(* CODESYS project Gateway_MLP_Validation.ecp

Project tree, tasks and I/O mapping:
  Steuerung : 750-8202 PFC200 2ETH RS, WAGO, order no. 0750-8202, version 5.15.4.20
    application Application
      libraries: ; Energy Edge Library, 3.5.16.10 (Zittau_Goerlitz University of Applied Sciences - IPM)
      task MLPinference (cyclic, interval 5 ms, priority 4) calls MLPinference
      Symbols
      program MLPinference [ST]
      function block WineTestMLP_3Layer [ST]
      function block WineTestMLP_2Layer [ST]
      function block WineTestMLP_1Layer [ST]
    Kbus : Kbus, WAGO, version 1.4.0.2
        unmapped channels: K-BUS diagnostics
    MODBUS
      MODBUS : MODBUS, WAGO, order no. n/a, version 1.1.1.15
    Serial
      COM1 : COM1, WAGO, version 0.0.0.19
*)

// Steuerung/Application/MLPinference
PROGRAM MLPinference
VAR
	// Seperate Inputs, since writen on MLP inputs via OPC UA fails

	inMLP1: ARRAY[1..11] OF REAL;
	inMLP2: ARRAY[1..11] OF REAL;	
	inMLP3: ARRAY[1..11] OF REAL;		

	MLP1: WineTestMLP_1Layer;
	MLP2: WineTestMLP_2Layer;
	MLP3: WineTestMLP_3Layer;
	
	recalculate: BOOL:=False;

END_VAR

IF recalculate THEN
	MLP1(in_1:=inMLP1[1], in_2:=inMLP1[2], in_3:=inMLP1[3], in_4:=inMLP1[4],
         in_5:=inMLP1[5], in_6:=inMLP1[6], in_7:=inMLP1[7], in_8:=inMLP1[8],
         in_9:=inMLP1[9], in_10:=inMLP1[10], in_11:=inMLP1[11]);
	MLP2(in_1:=inMLP2[1], in_2:=inMLP2[2], in_3:=inMLP2[3], in_4:=inMLP2[4],
         in_5:=inMLP2[5], in_6:=inMLP2[6], in_7:=inMLP2[7], in_8:=inMLP2[8],
         in_9:=inMLP2[9], in_10:=inMLP2[10], in_11:=inMLP2[11]);
	MLP3(in_1:=inMLP3[1], in_2:=inMLP3[2], in_3:=inMLP3[3], in_4:=inMLP3[4],
         in_5:=inMLP3[5], in_6:=inMLP3[6], in_7:=inMLP3[7], in_8:=inMLP3[8],
         in_9:=inMLP3[9], in_10:=inMLP3[10], in_11:=inMLP3[11]);
	recalculate := FALSE;
END_IF;

END_PROGRAM

// Steuerung/Application/WineTestMLP_1Layer
FUNCTION_BLOCK WineTestMLP_1Layer

VAR_INPUT
    in_1: REAL;
    in_2: REAL;
    in_3: REAL;
    in_4: REAL;
    in_5: REAL;
    in_6: REAL;
    in_7: REAL;
    in_8: REAL;
    in_9: REAL;
    in_10: REAL;
    in_11: REAL;
END_VAR

VAR
(* input array *)
    input: ARRAY[1..11] OF REAL;

(* hidden layer *)
(* Layer 1 *)
(* Neurons *)
    neuron_1_1: EEL.Neuron := (weights:=ADR(weights_1_1), bias:=(dw:=16#3f53bbb2), output:=0.0);
    neuron_1_2: EEL.Neuron := (weights:=ADR(weights_1_2), bias:=(dw:=16#3e774c91), output:=0.0);
    neuron_1_3: EEL.Neuron := (weights:=ADR(weights_1_3), bias:=(dw:=16#3f1b8655), output:=0.0);
    neuron_1_4: EEL.Neuron := (weights:=ADR(weights_1_4), bias:=(dw:=16#3f3931a5), output:=0.0);
    neuron_1_5: EEL.Neuron := (weights:=ADR(weights_1_5), bias:=(dw:=16#bd22504d), output:=0.0);
    neuron_1_6: EEL.Neuron := (weights:=ADR(weights_1_6), bias:=(dw:=16#3fcfd5a5), output:=0.0);
    neuron_1_7: EEL.Neuron := (weights:=ADR(weights_1_7), bias:=(dw:=16#3f154126), output:=0.0);
    neuron_1_8: EEL.Neuron := (weights:=ADR(weights_1_8), bias:=(dw:=16#bd8d8525), output:=0.0);
    neuron_1_9: EEL.Neuron := (weights:=ADR(weights_1_9), bias:=(dw:=16#3eede2e5), output:=0.0);
    neuron_1_10: EEL.Neuron := (weights:=ADR(weights_1_10), bias:=(dw:=16#bea8523e), output:=0.0);
    neuron_1_11: EEL.Neuron := (weights:=ADR(weights_1_11), bias:=(dw:=16#3f69af07), output:=0.0);
    neuron_1_12: EEL.Neuron := (weights:=ADR(weights_1_12), bias:=(dw:=16#3f1f30b5), output:=0.0);
    neuron_1_13: EEL.Neuron := (weights:=ADR(weights_1_13), bias:=(dw:=16#bc74c74c), output:=0.0);
    neuron_1_14: EEL.Neuron := (weights:=ADR(weights_1_14), bias:=(dw:=16#be4313a3), output:=0.0);
    neuron_1_15: EEL.Neuron := (weights:=ADR(weights_1_15), bias:=(dw:=16#bd1f8833), output:=0.0);
    neuron_1_16: EEL.Neuron := (weights:=ADR(weights_1_16), bias:=(dw:=16#3fa90598), output:=0.0);
    neuron_1_17: EEL.Neuron := (weights:=ADR(weights_1_17), bias:=(dw:=16#3f770b9d), output:=0.0);
    neuron_1_18: EEL.Neuron := (weights:=ADR(weights_1_18), bias:=(dw:=16#be4901f0), output:=0.0);
    neuron_1_19: EEL.Neuron := (weights:=ADR(weights_1_19), bias:=(dw:=16#bec4c956), output:=0.0);
    neuron_1_20: EEL.Neuron := (weights:=ADR(weights_1_20), bias:=(dw:=16#3effbf04), output:=0.0);
    neuron_1_21: EEL.Neuron := (weights:=ADR(weights_1_21), bias:=(dw:=16#3edacf42), output:=0.0);
    neuron_1_22: EEL.Neuron := (weights:=ADR(weights_1_22), bias:=(dw:=16#3f23897f), output:=0.0);
    neuron_1_23: EEL.Neuron := (weights:=ADR(weights_1_23), bias:=(dw:=16#bea09cbd), output:=0.0);
    neuron_1_24: EEL.Neuron := (weights:=ADR(weights_1_24), bias:=(dw:=16#3dabf729), output:=0.0);
    neuron_1_25: EEL.Neuron := (weights:=ADR(weights_1_25), bias:=(dw:=16#3f37b6a8), output:=0.0);
    hl_1_neurons: ARRAY[1..25] OF EEL.Neuron := [neuron_1_1, neuron_1_2, neuron_1_3, neuron_1_4, neuron_1_5, neuron_1_6, neuron_1_7, neuron_1_8, neuron_1_9, neuron_1_10, neuron_1_11, neuron_1_12, neuron_1_13, neuron_1_14, neuron_1_15, neuron_1_16, neuron_1_17, neuron_1_18, neuron_1_19, neuron_1_20, neuron_1_21, neuron_1_22, neuron_1_23, neuron_1_24, neuron_1_25];
(* Layer *)
    hidden_layer_1: EEL.Layer := (neurons:=ADR(hl_1_neurons), nNeurons:=25,activation:=12, threshold:=0.0);


    hlArray: ARRAY[1..1] of EEL.Layer := [hidden_layer_1];

(* output layer *)
    neuron_out_1: EEL.Neuron := (weights:=ADR(weights_out_1), bias:=(dw:=16#3ed09339), output:=0.0);
    out_neurons: ARRAY[1..1] OF EEL.Neuron := [neuron_out_1];
    out_layer: EEL.Layer := (neurons:=ADR(out_neurons), nNeurons:=1,activation:=3, threshold:=0.0);

(* MLP representation *)
    MLP: EEL.ANN := (input:=ADR(input), hidden:=ADR(hlArray), output:=ADR(out_layer), nInput:=11, nHidden:=1);
END_VAR

VAR_OUTPUT
    out_1: REAL;
END_VAR

VAR CONSTANT
    weights_1_1: ARRAY[1..11] OF EEL.dwREAL := [(dw:=16#bd130818), (dw:=16#3e57655a), (dw:=16#be872a61), (dw:=16#bcbdb356), (dw:=16#bd1f8b54), (dw:=16#3d854569), (dw:=16#bd02e86e), (dw:=16#3e87b72d), (dw:=16#3e9c4398), (dw:=16#3d24639f), (dw:=16#be22c6a0)];
    weights_1_2: ARRAY[1..11] OF EEL.dwREAL := [(dw:=16#3e2ba454), (dw:=16#bdc5c676), (dw:=16#3e3ef366), (dw:=16#3dcf9a7e), (dw:=16#bc0609b7), (dw:=16#3e3a72e8), (dw:=16#3e11846d), (dw:=16#3dc9d7ec), (dw:=16#bdd3251f), (dw:=16#389c9ec9), (dw:=16#3e24acb1)];
    weights_1_3: ARRAY[1..11] OF EEL.dwREAL := [(dw:=16#be00d314), (dw:=16#be382183), (dw:=16#3d07dd70), (dw:=16#bceefbce), (dw:=16#3dd44598), (dw:=16#3e1c33b7), (dw:=16#39f62b92), (dw:=16#bd632ec5), (dw:=16#3e1fecc7), (dw:=16#3c2fda30), (dw:=16#3d905dc3)];
    weights_1_4: ARRAY[1..11] OF EEL.dwREAL := [(dw:=16#bddbb524), (dw:=16#be554af8), (dw:=16#bda919bf), (dw:=16#3d3703ce), (dw:=16#3d70f66f), (dw:=16#bd44988d), (dw:=16#be1d6751), (dw:=16#bde58050), (dw:=16#3e51e712), (dw:=16#3d526bf5), (dw:=16#3e8ed860)];
    weights_1_5: ARRAY[1..11] OF EEL.dwREAL := [(dw:=16#3cbcb2b7), (dw:=16#bd2ecc57), (dw:=16#3de0a9a4), (dw:=16#3d298d90), (dw:=16#3dca6477), (dw:=16#bd4ba2ee), (dw:=16#3db50ce4), (dw:=16#3de32933), (dw:=16#bdead230), (dw:=16#3e2f56eb), (dw:=16#bd958376)];
    weights_1_6: ARRAY[1..11] OF EEL.dwREAL := [(dw:=16#bd8e9c27), (dw:=16#bd91e1fa), (dw:=16#bd6ca227), (dw:=16#3d671770), (dw:=16#bddaab27), (dw:=16#3dcc26e8), (dw:=16#3db16b56), (dw:=16#3d64df82), (dw:=16#bd0246ff), (dw:=16#bbc6cdd1), (dw:=16#3c404dc6)];
    weights_1_7: ARRAY[1..11] OF EEL.dwREAL := [(dw:=16#3bdecc96), (dw:=16#3bcbe5da), (dw:=16#3d2b50a4), (dw:=16#ba119a45), (dw:=16#bc438bf5), (dw:=16#3cb34be6), (dw:=16#bbc305c3), (dw:=16#bd0c3413), (dw:=16#bc8fb328), (dw:=16#3d39dc50), (dw:=16#bc19c7e9)];
    weights_1_8: ARRAY[1..11] OF EEL.dwREAL := [(dw:=16#bd61108b), (dw:=16#3d89d629), (dw:=16#bda47e84), (dw:=16#3cf8d9d7), (dw:=16#3d37cc3c), (dw:=16#3d57bf62), (dw:=16#3d606ad1), (dw:=16#bca8c762), (dw:=16#bd42dc34), (dw:=16#3e484431), (dw:=16#bc7633b2)];
    weights_1_9: ARRAY[1..11] OF EEL.dwREAL := [(dw:=16#be2c82e7), (dw:=16#3a1d1415), (dw:=16#bc41a5cf), (dw:=16#be42033e), (dw:=16#3dfcefe9), (dw:=16#be5ec4aa), (dw:=16#3e7ccf63), (dw:=16#be80d6a0), (dw:=16#3dd53c26), (dw:=16#bd937622), (dw:=16#be0c4531)];
    weights_1_10: ARRAY[1..11] OF EEL.dwREAL := [(dw:=16#be06776f), (dw:=16#3dffc8fc), (dw:=16#be17173a), (dw:=16#3d96ac7d), (dw:=16#3dcdc910), (dw:=16#3e4becaa), (dw:=16#3e05caf9), (dw:=16#3d694d95), (dw:=16#3e4c0015), (dw:=16#3e0131af), (dw:=16#bb05edc3)];
    weights_1_11: ARRAY[1..11] OF EEL.dwREAL := [(dw:=16#baaef3be), (dw:=16#be9ec245), (dw:=16#be0b5339), (dw:=16#3e006836), (dw:=16#bde8412e), (dw:=16#bb3055bf), (dw:=16#be01a90f), (dw:=16#3e01d2dd), (dw:=16#bce8fa64), (dw:=16#3e055065), (dw:=16#3e91930c)];
    weights_1_12: ARRAY[1..11] OF EEL.dwREAL := [(dw:=16#3df17f00), (dw:=16#bdb42e39), (dw:=16#3d769b38), (dw:=16#bdc2bb37), (dw:=16#be4bf9f7), (dw:=16#3e8e241d), (dw:=16#bd767810), (dw:=16#be4b11ea), (dw:=16#3d8e9dea), (dw:=16#bc47063f), (dw:=16#3e94287b)];
    weights_1_13: ARRAY[1..11] OF EEL.dwREAL := [(dw:=16#bc31da42), (dw:=16#bbaf341a), (dw:=16#bd287b58), (dw:=16#3c0e403d), (dw:=16#3d6f0f74), (dw:=16#3ccf2a99), (dw:=16#3d13f55d), (dw:=16#3b114489), (dw:=16#bd69e583), (dw:=16#3dccc3e8), (dw:=16#bc997423)];
    weights_1_14: ARRAY[1..11] OF EEL.dwREAL := [(dw:=16#3daef258), (dw:=16#be002661), (dw:=16#bc943066), (dw:=16#3db41f9b), (dw:=16#bb69810f), (dw:=16#3ca87ded), (dw:=16#3e3b0260), (dw:=16#3be476e7), (dw:=16#bdc6e2b0), (dw:=16#be2a7ec6), (dw:=16#3e3a9ab0)];
    weights_1_15: ARRAY[1..11] OF EEL.dwREAL := [(dw:=16#bd4de256), (dw:=16#3db57c57), (dw:=16#bdd2bb51), (dw:=16#3b9a972b), (dw:=16#bce2314f), (dw:=16#bb6dffbb), (dw:=16#bcc0e659), (dw:=16#3d149e41), (dw:=16#bdd52a52), (dw:=16#3e109b63), (dw:=16#bc04c6f8)];
    weights_1_16: ARRAY[1..11] OF EEL.dwREAL := [(dw:=16#3d8a3290), (dw:=16#3e05ee2b), (dw:=16#3d3b6ae0), (dw:=16#be0a58bd), (dw:=16#3dcb868a), (dw:=16#3c0cf723), (dw:=16#bde642cb), (dw:=16#bde659ca), (dw:=16#be364439), (dw:=16#3c9d0bf7), (dw:=16#be07452f)];
    weights_1_17: ARRAY[1..11] OF EEL.dwREAL := [(dw:=16#3d877279), (dw:=16#3e6a124c), (dw:=16#3d89c304), (dw:=16#3e07ed15), (dw:=16#3e252507), (dw:=16#be3de3f9), (dw:=16#be1dd184), (dw:=16#be851a24), (dw:=16#be94df33), (dw:=16#3e2c25ab), (dw:=16#3e250f69)];
    weights_1_18: ARRAY[1..11] OF EEL.dwREAL := [(dw:=16#bdeffadc), (dw:=16#bbd445cd), (dw:=16#bd498081), (dw:=16#3d837042), (dw:=16#bc6897bc), (dw:=16#be0bb273), (dw:=16#bdd77bed), (dw:=16#3c2604ab), (dw:=16#3e0991f3), (dw:=16#be4156f8), (dw:=16#3d8961a7)];
    weights_1_19: ARRAY[1..11] OF EEL.dwREAL := [(dw:=16#be60b820), (dw:=16#3e21be27), (dw:=16#bde0895a), (dw:=16#3c9ac8a0), (dw:=16#bdb6ab4f), (dw:=16#be2dbcf9), (dw:=16#be5d9323), (dw:=16#bd8e68dc), (dw:=16#3e2a844a), (dw:=16#beabbf6f), (dw:=16#3d7e7c9e)];
    weights_1_20: ARRAY[1..11] OF EEL.dwREAL := [(dw:=16#bdcd5501), (dw:=16#be35d7ff), (dw:=16#3e303c6a), (dw:=16#be29afe9), (dw:=16#be26862a), (dw:=16#be71656f), (dw:=16#bd35a65b), (dw:=16#3e7fae89), (dw:=16#be4008df), (dw:=16#3c073f38), (dw:=16#be4e845b)];
    weights_1_21: ARRAY[1..11] OF EEL.dwREAL := [(dw:=16#3d390b1c), (dw:=16#bd115fab), (dw:=16#3d306b93), (dw:=16#3c9372fd), (dw:=16#3b0bcc82), (dw:=16#3d0683fc), (dw:=16#bbe2c3af), (dw:=16#3c862552), (dw:=16#bd4d01b2), (dw:=16#3c988d92), (dw:=16#bd2800f4)];
    weights_1_22: ARRAY[1..11] OF EEL.dwREAL := [(dw:=16#bbcb6e7b), (dw:=16#3e93875e), (dw:=16#be8d8ad9), (dw:=16#3e3f7533), (dw:=16#bc0ee5ac), (dw:=16#be08c27e), (dw:=16#3eac5c4a), (dw:=16#bd94b032), (dw:=16#3e0d7cf5), (dw:=16#be485a5c), (dw:=16#bd07ce5c)];
    weights_1_23: ARRAY[1..11] OF EEL.dwREAL := [(dw:=16#bd559301), (dw:=16#be76dd4c), (dw:=16#bda748ba), (dw:=16#3cbe5fca), (dw:=16#bdd581e7), (dw:=16#3e196f17), (dw:=16#3d4f4331), (dw:=16#be4c92fd), (dw:=16#bca87a69), (dw:=16#be99c89d), (dw:=16#3de3a266)];
    weights_1_24: ARRAY[1..11] OF EEL.dwREAL := [(dw:=16#3ce204a2), (dw:=16#3d2ce670), (dw:=16#bd0e1f3b), (dw:=16#bde02636), (dw:=16#bd87123b), (dw:=16#bd6a8d42), (dw:=16#bde5a62f), (dw:=16#3c966757), (dw:=16#3dbb1b95), (dw:=16#be1fc696), (dw:=16#3bb752e5)];
    weights_1_25: ARRAY[1..11] OF EEL.dwREAL := [(dw:=16#3e3c38e9), (dw:=16#bd7c99d2), (dw:=16#3d16c39b), (dw:=16#bc866f5f), (dw:=16#3da78cfd), (dw:=16#bc07e312), (dw:=16#bdfa3ecf), (dw:=16#3decc2d5), (dw:=16#bd90452f), (dw:=16#3d867e23), (dw:=16#3d921418)];
    weights_out_1: ARRAY[1..25] OF EEL.dwREAL :=[(dw:=16#3f0bce82), (dw:=16#3ebc1fc3), (dw:=16#3eb9c571), (dw:=16#3eb97b27), (dw:=16#be8543b2), (dw:=16#3f11acc1), (dw:=16#3e4f512a), (dw:=16#be29c067), (dw:=16#3ecb8c44), (dw:=16#beba6d21), (dw:=16#3f3f28dc), (dw:=16#3f133968), (dw:=16#bdc67fed), (dw:=16#be9ae745), (dw:=16#be2c1060), (dw:=16#3f06b65f), (dw:=16#3f0c39f2), (dw:=16#be8ef089), (dw:=16#bf00858d), (dw:=16#3f01f92b), (dw:=16#3e15fc18), (dw:=16#3edc4104), (dw:=16#beeb452e), (dw:=16#be4c2559), (dw:=16#3e87fc13)];
END_VAR

(* get inputs *)
input[1] := in_1;
input[2] := in_2;
input[3] := in_3;
input[4] := in_4;
input[5] := in_5;
input[6] := in_6;
input[7] := in_7;
input[8] := in_8;
input[9] := in_9;
input[10] := in_10;
input[11] := in_11;

(* MLP inference *)
EEL.CallANN(ANN:=MLP);

(* set outputs *)
out_1 := out_neurons[1].output;

END_FUNCTION_BLOCK

// Steuerung/Application/WineTestMLP_2Layer
FUNCTION_BLOCK WineTestMLP_2Layer

VAR_INPUT
    in_1: REAL;
    in_2: REAL;
    in_3: REAL;
    in_4: REAL;
    in_5: REAL;
    in_6: REAL;
    in_7: REAL;
    in_8: REAL;
    in_9: REAL;
    in_10: REAL;
    in_11: REAL;
END_VAR

VAR
(* input array *)
    input: ARRAY[1..11] OF REAL;

(* hidden layer *)
(* Layer 1 *)
(* Neurons *)
    neuron_1_1: EEL.Neuron := (weights:=ADR(weights_1_1), bias:=(dw:=16#3c825e3d), output:=0.0);
    neuron_1_2: EEL.Neuron := (weights:=ADR(weights_1_2), bias:=(dw:=16#bea43e80), output:=0.0);
    neuron_1_3: EEL.Neuron := (weights:=ADR(weights_1_3), bias:=(dw:=16#be707efb), output:=0.0);
    neuron_1_4: EEL.Neuron := (weights:=ADR(weights_1_4), bias:=(dw:=16#3e146b2a), output:=0.0);
    neuron_1_5: EEL.Neuron := (weights:=ADR(weights_1_5), bias:=(dw:=16#3f5269ab), output:=0.0);
    neuron_1_6: EEL.Neuron := (weights:=ADR(weights_1_6), bias:=(dw:=16#3f4f3302), output:=0.0);
    neuron_1_7: EEL.Neuron := (weights:=ADR(weights_1_7), bias:=(dw:=16#3f42e11b), output:=0.0);
    neuron_1_8: EEL.Neuron := (weights:=ADR(weights_1_8), bias:=(dw:=16#3f40ae65), output:=0.0);
    neuron_1_9: EEL.Neuron := (weights:=ADR(weights_1_9), bias:=(dw:=16#be83203b), output:=0.0);
    neuron_1_10: EEL.Neuron := (weights:=ADR(weights_1_10), bias:=(dw:=16#bea2b30d), output:=0.0);
    neuron_1_11: EEL.Neuron := (weights:=ADR(weights_1_11), bias:=(dw:=16#3f3500ff), output:=0.0);
    neuron_1_12: EEL.Neuron := (weights:=ADR(weights_1_12), bias:=(dw:=16#3eb84acd), output:=0.0);
    neuron_1_13: EEL.Neuron := (weights:=ADR(weights_1_13), bias:=(dw:=16#3f335357), output:=0.0);
    neuron_1_14: EEL.Neuron := (weights:=ADR(weights_1_14), bias:=(dw:=16#bdd40d48), output:=0.0);
    neuron_1_15: EEL.Neuron := (weights:=ADR(weights_1_15), bias:=(dw:=16#bd81df84), output:=0.0);
    neuron_1_16: EEL.Neuron := (weights:=ADR(weights_1_16), bias:=(dw:=16#bddf6ef8), output:=0.0);
    neuron_1_17: EEL.Neuron := (weights:=ADR(weights_1_17), bias:=(dw:=16#3e36da12), output:=0.0);
    neuron_1_18: EEL.Neuron := (weights:=ADR(weights_1_18), bias:=(dw:=16#3f045953), output:=0.0);
    neuron_1_19: EEL.Neuron := (weights:=ADR(weights_1_19), bias:=(dw:=16#3ed228f5), output:=0.0);
    neuron_1_20: EEL.Neuron := (weights:=ADR(weights_1_20), bias:=(dw:=16#3ed4b31e), output:=0.0);
    neuron_1_21: EEL.Neuron := (weights:=ADR(weights_1_21), bias:=(dw:=16#bde4ea74), output:=0.0);
    neuron_1_22: EEL.Neuron := (weights:=ADR(weights_1_22), bias:=(dw:=16#3ec57342), output:=0.0);
    neuron_1_23: EEL.Neuron := (weights:=ADR(weights_1_23), bias:=(dw:=16#3d34d29b), output:=0.0);
    neuron_1_24: EEL.Neuron := (weights:=ADR(weights_1_24), bias:=(dw:=16#3f80457c), output:=0.0);
    neuron_1_25: EEL.Neuron := (weights:=ADR(weights_1_25), bias:=(dw:=16#bdaa519e), output:=0.0);
    hl_1_neurons: ARRAY[1..25] OF EEL.Neuron := [neuron_1_1, neuron_1_2, neuron_1_3, neuron_1_4, neuron_1_5, neuron_1_6, neuron_1_7, neuron_1_8, neuron_1_9, neuron_1_10, neuron_1_11, neuron_1_12, neuron_1_13, neuron_1_14, neuron_1_15, neuron_1_16, neuron_1_17, neuron_1_18, neuron_1_19, neuron_1_20, neuron_1_21, neuron_1_22, neuron_1_23, neuron_1_24, neuron_1_25];
(* Layer *)
    hidden_layer_1: EEL.Layer := (neurons:=ADR(hl_1_neurons), nNeurons:=25,activation:=12, threshold:=0.0);

(* Layer 2 *)
(* Neurons *)
    neuron_2_1: EEL.Neuron := (weights:=ADR(weights_2_1), bias:=(dw:=16#bf209498), output:=0.0);
    neuron_2_2: EEL.Neuron := (weights:=ADR(weights_2_2), bias:=(dw:=16#beeab10d), output:=0.0);
    neuron_2_3: EEL.Neuron := (weights:=ADR(weights_2_3), bias:=(dw:=16#3f4d4c49), output:=0.0);
    neuron_2_4: EEL.Neuron := (weights:=ADR(weights_2_4), bias:=(dw:=16#3f306120), output:=0.0);
    neuron_2_5: EEL.Neuron := (weights:=ADR(weights_2_5), bias:=(dw:=16#3f02efd6), output:=0.0);
    hl_2_neurons: ARRAY[1..5] OF EEL.Neuron := [neuron_2_1, neuron_2_2, neuron_2_3, neuron_2_4, neuron_2_5];
(* Layer *)
    hidden_layer_2: EEL.Layer := (neurons:=ADR(hl_2_neurons), nNeurons:=5,activation:=12, threshold:=0.0);


    hlArray: ARRAY[1..2] of EEL.Layer := [hidden_layer_1, hidden_layer_2];

(* output layer *)
    neuron_out_1: EEL.Neuron := (weights:=ADR(weights_out_1), bias:=(dw:=16#3d255e43), output:=0.0);
    out_neurons: ARRAY[1..1] OF EEL.Neuron := [neuron_out_1];
    out_layer: EEL.Layer := (neurons:=ADR(out_neurons), nNeurons:=1,activation:=3, threshold:=0.0);

(* MLP representation *)
    MLP: EEL.ANN := (input:=ADR(input), hidden:=ADR(hlArray), output:=ADR(out_layer), nInput:=11, nHidden:=2);
END_VAR

VAR_OUTPUT
    out_1: REAL;
END_VAR

VAR CONSTANT
    weights_1_1: ARRAY[1..11] OF EEL.dwREAL := [(dw:=16#3c55f395), (dw:=16#3d97f889), (dw:=16#bdf2c0f1), (dw:=16#bd2fd6c7), (dw:=16#bb6cef76), (dw:=16#3cf182be), (dw:=16#bd105294), (dw:=16#3d93a886), (dw:=16#3dc68841), (dw:=16#3d14c557), (dw:=16#bde70111)];
    weights_1_2: ARRAY[1..11] OF EEL.dwREAL := [(dw:=16#3c87590b), (dw:=16#be179a25), (dw:=16#3dbbbc1f), (dw:=16#3df58434), (dw:=16#bb86d268), (dw:=16#3d6793f4), (dw:=16#3e2f66db), (dw:=16#bc1c4752), (dw:=16#bd771fa5), (dw:=16#3c9d340b), (dw:=16#3e2e124a)];
    weights_1_3: ARRAY[1..11] OF EEL.dwREAL := [(dw:=16#be1928ea), (dw:=16#bcb78dd7), (dw:=16#be1abcc7), (dw:=16#3cc4fb9c), (dw:=16#3e3e9e8c), (dw:=16#3dd5666e), (dw:=16#3e2c61fa), (dw:=16#bc51bda6), (dw:=16#bc0213e6), (dw:=16#3e843141), (dw:=16#bd86a7cd)];
    weights_1_4: ARRAY[1..11] OF EEL.dwREAL := [(dw:=16#bde9f6b3), (dw:=16#be864c9d), (dw:=16#bdd7d352), (dw:=16#3ddbbce3), (dw:=16#bd9425e1), (dw:=16#be54217c), (dw:=16#be8b1d76), (dw:=16#bead0200), (dw:=16#3e080905), (dw:=16#3e4c7713), (dw:=16#3edcc87a)];
    weights_1_5: ARRAY[1..11] OF EEL.dwREAL := [(dw:=16#be335363), (dw:=16#3e8dc1ea), (dw:=16#be03a942), (dw:=16#3bcf609d), (dw:=16#3e1897e6), (dw:=16#be4bf5fc), (dw:=16#bcd23276), (dw:=16#be42dff3), (dw:=16#3d43abaf), (dw:=16#393a1b60), (dw:=16#3d785a49)];
    weights_1_6: ARRAY[1..11] OF EEL.dwREAL := [(dw:=16#be68d82a), (dw:=16#beb24ff3), (dw:=16#be809d52), (dw:=16#3d7e0e21), (dw:=16#3d8c82b6), (dw:=16#3d8439d6), (dw:=16#3de6bfc8), (dw:=16#3ce42630), (dw:=16#3df1c506), (dw:=16#bcfe46e6), (dw:=16#3dd0b2e3)];
    weights_1_7: ARRAY[1..11] OF EEL.dwREAL := [(dw:=16#bd8380e9), (dw:=16#be236a44), (dw:=16#3d6edae9), (dw:=16#3c45e317), (dw:=16#be9600ec), (dw:=16#3ea9a652), (dw:=16#bdff09bb), (dw:=16#be020921), (dw:=16#3d982899), (dw:=16#3ccea5e6), (dw:=16#3d59e16e)];
    weights_1_8: ARRAY[1..11] OF EEL.dwREAL := [(dw:=16#bda79eeb), (dw:=16#3ea1e6a9), (dw:=16#bea6ce7e), (dw:=16#3ddaa327), (dw:=16#3d912ea1), (dw:=16#3d207bd8), (dw:=16#3e4656a9), (dw:=16#3e5dbe2c), (dw:=16#3e3c3b0c), (dw:=16#bd77e2b6), (dw:=16#bdcd1367)];
    weights_1_9: ARRAY[1..11] OF EEL.dwREAL := [(dw:=16#bdfddd3c), (dw:=16#bd3512f9), (dw:=16#3c7e1a12), (dw:=16#3d943969), (dw:=16#bdb791d3), (dw:=16#be76dc3b), (dw:=16#be27a5c5), (dw:=16#bdee2a46), (dw:=16#3ea17800), (dw:=16#be91ac3b), (dw:=16#3d9e6bc0)];
    weights_1_10: ARRAY[1..11] OF EEL.dwREAL := [(dw:=16#3c573eb3), (dw:=16#3e0a5e57), (dw:=16#be150f11), (dw:=16#3d8d8eaf), (dw:=16#3e45f997), (dw:=16#3e2366de), (dw:=16#3e17fd0a), (dw:=16#3d3be255), (dw:=16#3e7ed11c), (dw:=16#bdd5be10), (dw:=16#bc19a00c)];
    weights_1_11: ARRAY[1..11] OF EEL.dwREAL := [(dw:=16#3e36c9ed), (dw:=16#be3b9a59), (dw:=16#be4038ca), (dw:=16#3d983102), (dw:=16#bd8edfc8), (dw:=16#bda9d3ca), (dw:=16#be919aa3), (dw:=16#3d3c3e2f), (dw:=16#be4dba64), (dw:=16#3e3da2a3), (dw:=16#3e70ae22)];
    weights_1_12: ARRAY[1..11] OF EEL.dwREAL := [(dw:=16#3d127e5a), (dw:=16#3e54ca31), (dw:=16#bdd629f5), (dw:=16#bdbe7362), (dw:=16#be4dca3b), (dw:=16#3e8746cc), (dw:=16#3d4740bb), (dw:=16#be6cae03), (dw:=16#3ea4f6dd), (dw:=16#be6f5147), (dw:=16#3e172058)];
    weights_1_13: ARRAY[1..11] OF EEL.dwREAL := [(dw:=16#bda4d07c), (dw:=16#3dd4e381), (dw:=16#3e2d5f2b), (dw:=16#3e51414f), (dw:=16#3e38e62f), (dw:=16#bd811133), (dw:=16#3d8593f5), (dw:=16#bb7ee211), (dw:=16#be8c3e0c), (dw:=16#3d5430be), (dw:=16#3eb6e43f)];
    weights_1_14: ARRAY[1..11] OF EEL.dwREAL := [(dw:=16#3d087928), (dw:=16#be588505), (dw:=16#bd9fed10), (dw:=16#3c1a81fe), (dw:=16#3bbda7de), (dw:=16#3d7835c4), (dw:=16#3da6ad88), (dw:=16#bddb6be4), (dw:=16#bd8dff7c), (dw:=16#be9a0b17), (dw:=16#3e155c9f)];
    weights_1_15: ARRAY[1..11] OF EEL.dwREAL := [(dw:=16#be9634d6), (dw:=16#3df0cb56), (dw:=16#be1c364d), (dw:=16#3d9df541), (dw:=16#be2a9506), (dw:=16#3d460d83), (dw:=16#bdc01b09), (dw:=16#3e299911), (dw:=16#bdfdd8a3), (dw:=16#3a0e045c), (dw:=16#3dd5b3a1)];
    weights_1_16: ARRAY[1..11] OF EEL.dwREAL := [(dw:=16#3d68eef2), (dw:=16#3e3d0509), (dw:=16#3d42ec27), (dw:=16#bd429b4e), (dw:=16#bd0a176f), (dw:=16#b9a0af16), (dw:=16#be1116e7), (dw:=16#3cb7164d), (dw:=16#3dd2fe3b), (dw:=16#be69bec8), (dw:=16#bc0d99d3)];
    weights_1_17: ARRAY[1..11] OF EEL.dwREAL := [(dw:=16#3ac5955e), (dw:=16#3d65b091), (dw:=16#ba967171), (dw:=16#3d2189d9), (dw:=16#3c86d532), (dw:=16#bd34aab0), (dw:=16#bd7ce1f5), (dw:=16#bd292a56), (dw:=16#bd55562a), (dw:=16#3d2e975a), (dw:=16#3c8e27b4)];
    weights_1_18: ARRAY[1..11] OF EEL.dwREAL := [(dw:=16#3e0895f2), (dw:=16#be5dc128), (dw:=16#3db85118), (dw:=16#bd9e7564), (dw:=16#3db12341), (dw:=16#bdfe9a1f), (dw:=16#bd9ab688), (dw:=16#3da42ef1), (dw:=16#3d1b8ff7), (dw:=16#3d1c2cf2), (dw:=16#bc32ab5e)];
    weights_1_19: ARRAY[1..11] OF EEL.dwREAL := [(dw:=16#be03d672), (dw:=16#3e3246c9), (dw:=16#3b904917), (dw:=16#bd7ce276), (dw:=16#3d2ce7c6), (dw:=16#be3b78ec), (dw:=16#3de4e257), (dw:=16#3e4cbd93), (dw:=16#3e237ea6), (dw:=16#be217033), (dw:=16#be596151)];
    weights_1_20: ARRAY[1..11] OF EEL.dwREAL := [(dw:=16#bc8a9c87), (dw:=16#be8bb8ff), (dw:=16#3e034b20), (dw:=16#be0f26bb), (dw:=16#be0cab67), (dw:=16#be51f1c9), (dw:=16#bd14e375), (dw:=16#3e4d9e7c), (dw:=16#be7facca), (dw:=16#3d9ac88f), (dw:=16#bdc66fdb)];
    weights_1_21: ARRAY[1..11] OF EEL.dwREAL := [(dw:=16#3ddd3515), (dw:=16#bc063c7f), (dw:=16#3e25e617), (dw:=16#bc13eb3f), (dw:=16#3b5297ce), (dw:=16#bd9ec959), (dw:=16#bc45d03b), (dw:=16#3dd84793), (dw:=16#bcc572a7), (dw:=16#bc10e2a3), (dw:=16#bc197ebe)];
    weights_1_22: ARRAY[1..11] OF EEL.dwREAL := [(dw:=16#3d305014), (dw:=16#3ce9a43b), (dw:=16#be5d702d), (dw:=16#bdbc0cc8), (dw:=16#bdc0fb4f), (dw:=16#be38949c), (dw:=16#3e1294fc), (dw:=16#be4bd803), (dw:=16#bdc1130c), (dw:=16#bd2abf84), (dw:=16#be2b7d08)];
    weights_1_23: ARRAY[1..11] OF EEL.dwREAL := [(dw:=16#be1572db), (dw:=16#be611c59), (dw:=16#be5d49e3), (dw:=16#bd8383ef), (dw:=16#be45f680), (dw:=16#3e7057cc), (dw:=16#3de87245), (dw:=16#be371554), (dw:=16#be32cd05), (dw:=16#bd9b822b), (dw:=16#bbed6728)];
    weights_1_24: ARRAY[1..11] OF EEL.dwREAL := [(dw:=16#3e96f08a), (dw:=16#bdfebc24), (dw:=16#3e853f97), (dw:=16#be114e5d), (dw:=16#bd9775d3), (dw:=16#3dfc2c40), (dw:=16#be43448c), (dw:=16#3dc08573), (dw:=16#3d488d25), (dw:=16#3db4143b), (dw:=16#bdd129ac)];
    weights_1_25: ARRAY[1..11] OF EEL.dwREAL := [(dw:=16#3dd4b883), (dw:=16#bdafdffd), (dw:=16#3df40f53), (dw:=16#3d926627), (dw:=16#3df30f03), (dw:=16#be16e92a), (dw:=16#3d9cce80), (dw:=16#3e2dfeb4), (dw:=16#bd50fb60), (dw:=16#3e529d57), (dw:=16#bc053847)];
    weights_2_1: ARRAY[1..25] OF EEL.dwREAL := [(dw:=16#3db52b5f), (dw:=16#3e2eb117), (dw:=16#3dbe5ef2), (dw:=16#3e48ef28), (dw:=16#bddccc99), (dw:=16#3d84f99a), (dw:=16#3d533b86), (dw:=16#3e050ffd), (dw:=16#3e717c19), (dw:=16#3e052471), (dw:=16#3bc1b843), (dw:=16#3e708f26), (dw:=16#3dd2f5cb), (dw:=16#3e4c7dad), (dw:=16#3e49f8b0), (dw:=16#3e29f24d), (dw:=16#bcb3fe63), (dw:=16#3da73504), (dw:=16#3e89a4f1), (dw:=16#3e114061), (dw:=16#3e3567ee), (dw:=16#bd1e8f1b), (dw:=16#3e8a5f7f), (dw:=16#3bf97a15), (dw:=16#3de3548d)];
    weights_2_2: ARRAY[1..25] OF EEL.dwREAL := [(dw:=16#3d9ff412), (dw:=16#3c0a38f9), (dw:=16#3d6fc6ce), (dw:=16#3d8219c8), (dw:=16#3c831752), (dw:=16#bcda3fe6), (dw:=16#3d9fb4e8), (dw:=16#3d044e55), (dw:=16#3cd0bfb1), (dw:=16#3c410d41), (dw:=16#3d141591), (dw:=16#3da9fbb0), (dw:=16#3cb962c4), (dw:=16#3d53588a), (dw:=16#bcd5ccab), (dw:=16#3cc456ae), (dw:=16#3b4bb5a9), (dw:=16#3d355cf9), (dw:=16#3d761043), (dw:=16#3c1f2cb5), (dw:=16#3cedef62), (dw:=16#bb2463b1), (dw:=16#3ce08616), (dw:=16#3de670ac), (dw:=16#bc6007cc)];
    weights_2_3: ARRAY[1..25] OF EEL.dwREAL := [(dw:=16#3d4cb90a), (dw:=16#bdde7c82), (dw:=16#be01497b), (dw:=16#bd94dcb5), (dw:=16#3e2881ac), (dw:=16#3e9d7c24), (dw:=16#3dcc19f7), (dw:=16#3ec5a4dd), (dw:=16#be27da0e), (dw:=16#bdbcd37f), (dw:=16#3e134bbb), (dw:=16#bda97198), (dw:=16#3eaa0fc0), (dw:=16#be033269), (dw:=16#be096700), (dw:=16#bddc3393), (dw:=16#3e11c485), (dw:=16#3e01bb1c), (dw:=16#3d304485), (dw:=16#3e513004), (dw:=16#be3b2e4d), (dw:=16#3e0451a0), (dw:=16#bd6cf0db), (dw:=16#3e930b90), (dw:=16#be805a08)];
    weights_2_4: ARRAY[1..25] OF EEL.dwREAL := [(dw:=16#b9d452f8), (dw:=16#be1a7fab), (dw:=16#be4787b6), (dw:=16#bdedf2a7), (dw:=16#3e625c96), (dw:=16#3ea5625d), (dw:=16#3e74668c), (dw:=16#3ec10889), (dw:=16#be6f00b4), (dw:=16#bdf1b4b1), (dw:=16#3e63e5b3), (dw:=16#bd596a02), (dw:=16#3e4586ad), (dw:=16#be41a5a8), (dw:=16#be1285de), (dw:=16#be2157ae), (dw:=16#3d174f89), (dw:=16#bc7afe67), (dw:=16#bd87b196), (dw:=16#3d625f0e), (dw:=16#bd82816c), (dw:=16#3e04b44f), (dw:=16#be40b546), (dw:=16#3f095b7c), (dw:=16#be9ec030)];
    weights_2_5: ARRAY[1..25] OF EEL.dwREAL := [(dw:=16#bdc99a8c), (dw:=16#bdc89b92), (dw:=16#be2f307e), (dw:=16#3ee62477), (dw:=16#3e987693), (dw:=16#3ebf61a1), (dw:=16#3eed7efb), (dw:=16#3e95a161), (dw:=16#bea72881), (dw:=16#be9f734f), (dw:=16#3eb9ae24), (dw:=16#3f054924), (dw:=16#3f1d93b6), (dw:=16#be47877a), (dw:=16#be87bd9a), (dw:=16#be259c5d), (dw:=16#bd369f68), (dw:=16#3e8014a5), (dw:=16#3ea39572), (dw:=16#3e7c1521), (dw:=16#3de38f47), (dw:=16#3e68cf83), (dw:=16#3e86a42e), (dw:=16#3ec884b7), (dw:=16#3de4f387)];
    weights_out_1: ARRAY[1..5] OF EEL.dwREAL :=[(dw:=16#bf23d55d), (dw:=16#bdaa1c3e), (dw:=16#3ee49b6b), (dw:=16#3f20ca2e), (dw:=16#3f66b142)];
END_VAR

(* get inputs *)
input[1] := in_1;
input[2] := in_2;
input[3] := in_3;
input[4] := in_4;
input[5] := in_5;
input[6] := in_6;
input[7] := in_7;
input[8] := in_8;
input[9] := in_9;
input[10] := in_10;
input[11] := in_11;

(* MLP inference *)
EEL.CallANN(ANN:=MLP);

(* set outputs *)
out_1 := out_neurons[1].output;

END_FUNCTION_BLOCK

// Steuerung/Application/WineTestMLP_3Layer
FUNCTION_BLOCK WineTestMLP_3Layer

VAR_INPUT
    in_1: REAL;
    in_2: REAL;
    in_3: REAL;
    in_4: REAL;
    in_5: REAL;
    in_6: REAL;
    in_7: REAL;
    in_8: REAL;
    in_9: REAL;
    in_10: REAL;
    in_11: REAL;
END_VAR

VAR
(* input array *)
    input: ARRAY[1..11] OF REAL;

(* hidden layer *)
(* Layer 1 *)
(* Neurons *)
    neuron_1_1: EEL.Neuron := (weights:=ADR(weights_1_1), bias:=(dw:=16#3f08ef92), output:=0.0);
    neuron_1_2: EEL.Neuron := (weights:=ADR(weights_1_2), bias:=(dw:=16#bdca5113), output:=0.0);
    neuron_1_3: EEL.Neuron := (weights:=ADR(weights_1_3), bias:=(dw:=16#3e68de37), output:=0.0);
    neuron_1_4: EEL.Neuron := (weights:=ADR(weights_1_4), bias:=(dw:=16#3d6e3327), output:=0.0);
    neuron_1_5: EEL.Neuron := (weights:=ADR(weights_1_5), bias:=(dw:=16#3d1d484a), output:=0.0);
    neuron_1_6: EEL.Neuron := (weights:=ADR(weights_1_6), bias:=(dw:=16#3f184f59), output:=0.0);
    neuron_1_7: EEL.Neuron := (weights:=ADR(weights_1_7), bias:=(dw:=16#3f1b7a91), output:=0.0);
    neuron_1_8: EEL.Neuron := (weights:=ADR(weights_1_8), bias:=(dw:=16#3edb027e), output:=0.0);
    neuron_1_9: EEL.Neuron := (weights:=ADR(weights_1_9), bias:=(dw:=16#3d189d54), output:=0.0);
    neuron_1_10: EEL.Neuron := (weights:=ADR(weights_1_10), bias:=(dw:=16#3d5c6ba9), output:=0.0);
    neuron_1_11: EEL.Neuron := (weights:=ADR(weights_1_11), bias:=(dw:=16#3f39ab73), output:=0.0);
    neuron_1_12: EEL.Neuron := (weights:=ADR(weights_1_12), bias:=(dw:=16#3e6b760a), output:=0.0);
    neuron_1_13: EEL.Neuron := (weights:=ADR(weights_1_13), bias:=(dw:=16#3f0cf376), output:=0.0);
    neuron_1_14: EEL.Neuron := (weights:=ADR(weights_1_14), bias:=(dw:=16#3ea1b992), output:=0.0);
    neuron_1_15: EEL.Neuron := (weights:=ADR(weights_1_15), bias:=(dw:=16#3d8152bd), output:=0.0);
    neuron_1_16: EEL.Neuron := (weights:=ADR(weights_1_16), bias:=(dw:=16#3eadaf4c), output:=0.0);
    neuron_1_17: EEL.Neuron := (weights:=ADR(weights_1_17), bias:=(dw:=16#3f56b40e), output:=0.0);
    neuron_1_18: EEL.Neuron := (weights:=ADR(weights_1_18), bias:=(dw:=16#3efdcac9), output:=0.0);
    neuron_1_19: EEL.Neuron := (weights:=ADR(weights_1_19), bias:=(dw:=16#3e9a8ca0), output:=0.0);
    neuron_1_20: EEL.Neuron := (weights:=ADR(weights_1_20), bias:=(dw:=16#3d5f9176), output:=0.0);
    neuron_1_21: EEL.Neuron := (weights:=ADR(weights_1_21), bias:=(dw:=16#bd9f8478), output:=0.0);
    neuron_1_22: EEL.Neuron := (weights:=ADR(weights_1_22), bias:=(dw:=16#bef177ac), output:=0.0);
    neuron_1_23: EEL.Neuron := (weights:=ADR(weights_1_23), bias:=(dw:=16#bd743fb7), output:=0.0);
    neuron_1_24: EEL.Neuron := (weights:=ADR(weights_1_24), bias:=(dw:=16#3f450ace), output:=0.0);
    neuron_1_25: EEL.Neuron := (weights:=ADR(weights_1_25), bias:=(dw:=16#be562e07), output:=0.0);
    hl_1_neurons: ARRAY[1..25] OF EEL.Neuron := [neuron_1_1, neuron_1_2, neuron_1_3, neuron_1_4, neuron_1_5, neuron_1_6, neuron_1_7, neuron_1_8, neuron_1_9, neuron_1_10, neuron_1_11, neuron_1_12, neuron_1_13, neuron_1_14, neuron_1_15, neuron_1_16, neuron_1_17, neuron_1_18, neuron_1_19, neuron_1_20, neuron_1_21, neuron_1_22, neuron_1_23, neuron_1_24, neuron_1_25];
(* Layer *)
    hidden_layer_1: EEL.Layer := (neurons:=ADR(hl_1_neurons), nNeurons:=25,activation:=12, threshold:=0.0);

(* Layer 2 *)
(* Neurons *)
    neuron_2_1: EEL.Neuron := (weights:=ADR(weights_2_1), bias:=(dw:=16#bf08b91c), output:=0.0);
    neuron_2_2: EEL.Neuron := (weights:=ADR(weights_2_2), bias:=(dw:=16#be00d19c), output:=0.0);
    neuron_2_3: EEL.Neuron := (weights:=ADR(weights_2_3), bias:=(dw:=16#3f2e5438), output:=0.0);
    neuron_2_4: EEL.Neuron := (weights:=ADR(weights_2_4), bias:=(dw:=16#3e61c3dd), output:=0.0);
    neuron_2_5: EEL.Neuron := (weights:=ADR(weights_2_5), bias:=(dw:=16#3df739b3), output:=0.0);
    hl_2_neurons: ARRAY[1..5] OF EEL.Neuron := [neuron_2_1, neuron_2_2, neuron_2_3, neuron_2_4, neuron_2_5];
(* Layer *)
    hidden_layer_2: EEL.Layer := (neurons:=ADR(hl_2_neurons), nNeurons:=5,activation:=12, threshold:=0.0);

(* Layer 3 *)
(* Neurons *)
    neuron_3_1: EEL.Neuron := (weights:=ADR(weights_3_1), bias:=(dw:=16#3ec7482b), output:=0.0);
    neuron_3_2: EEL.Neuron := (weights:=ADR(weights_3_2), bias:=(dw:=16#bcd6b239), output:=0.0);
    neuron_3_3: EEL.Neuron := (weights:=ADR(weights_3_3), bias:=(dw:=16#3f23d06f), output:=0.0);
    neuron_3_4: EEL.Neuron := (weights:=ADR(weights_3_4), bias:=(dw:=16#3eeeb131), output:=0.0);
    neuron_3_5: EEL.Neuron := (weights:=ADR(weights_3_5), bias:=(dw:=16#3e44f054), output:=0.0);
    neuron_3_6: EEL.Neuron := (weights:=ADR(weights_3_6), bias:=(dw:=16#3c95a37d), output:=0.0);
    neuron_3_7: EEL.Neuron := (weights:=ADR(weights_3_7), bias:=(dw:=16#3ee20e82), output:=0.0);
    neuron_3_8: EEL.Neuron := (weights:=ADR(weights_3_8), bias:=(dw:=16#3e6660c5), output:=0.0);
    neuron_3_9: EEL.Neuron := (weights:=ADR(weights_3_9), bias:=(dw:=16#bec740bb), output:=0.0);
    neuron_3_10: EEL.Neuron := (weights:=ADR(weights_3_10), bias:=(dw:=16#be2f1769), output:=0.0);
    neuron_3_11: EEL.Neuron := (weights:=ADR(weights_3_11), bias:=(dw:=16#bd211747), output:=0.0);
    neuron_3_12: EEL.Neuron := (weights:=ADR(weights_3_12), bias:=(dw:=16#3ef925de), output:=0.0);
    neuron_3_13: EEL.Neuron := (weights:=ADR(weights_3_13), bias:=(dw:=16#3cbac84a), output:=0.0);
    neuron_3_14: EEL.Neuron := (weights:=ADR(weights_3_14), bias:=(dw:=16#bd971787), output:=0.0);
    neuron_3_15: EEL.Neuron := (weights:=ADR(weights_3_15), bias:=(dw:=16#bde24186), output:=0.0);
    neuron_3_16: EEL.Neuron := (weights:=ADR(weights_3_16), bias:=(dw:=16#bef55d88), output:=0.0);
    neuron_3_17: EEL.Neuron := (weights:=ADR(weights_3_17), bias:=(dw:=16#3ec551eb), output:=0.0);
    neuron_3_18: EEL.Neuron := (weights:=ADR(weights_3_18), bias:=(dw:=16#be2ab042), output:=0.0);
    neuron_3_19: EEL.Neuron := (weights:=ADR(weights_3_19), bias:=(dw:=16#3f2aaa3d), output:=0.0);
    neuron_3_20: EEL.Neuron := (weights:=ADR(weights_3_20), bias:=(dw:=16#be8c5896), output:=0.0);
    hl_3_neurons: ARRAY[1..20] OF EEL.Neuron := [neuron_3_1, neuron_3_2, neuron_3_3, neuron_3_4, neuron_3_5, neuron_3_6, neuron_3_7, neuron_3_8, neuron_3_9, neuron_3_10, neuron_3_11, neuron_3_12, neuron_3_13, neuron_3_14, neuron_3_15, neuron_3_16, neuron_3_17, neuron_3_18, neuron_3_19, neuron_3_20];
(* Layer *)
    hidden_layer_3: EEL.Layer := (neurons:=ADR(hl_3_neurons), nNeurons:=20,activation:=12, threshold:=0.0);


    hlArray: ARRAY[1..3] of EEL.Layer := [hidden_layer_1, hidden_layer_2, hidden_layer_3];

(* output layer *)
    neuron_out_1: EEL.Neuron := (weights:=ADR(weights_out_1), bias:=(dw:=16#3e0c0c0f), output:=0.0);
    out_neurons: ARRAY[1..1] OF EEL.Neuron := [neuron_out_1];
    out_layer: EEL.Layer := (neurons:=ADR(out_neurons), nNeurons:=1,activation:=3, threshold:=0.0);

(* MLP representation *)
    MLP: EEL.ANN := (input:=ADR(input), hidden:=ADR(hlArray), output:=ADR(out_layer), nInput:=11, nHidden:=3);
END_VAR

VAR_OUTPUT
    out_1: REAL;
END_VAR

VAR CONSTANT
    weights_1_1: ARRAY[1..11] OF EEL.dwREAL := [(dw:=16#bc88b305), (dw:=16#3e1c048f), (dw:=16#be5b562c), (dw:=16#bd9a0710), (dw:=16#bdd644d8), (dw:=16#3d203cbb), (dw:=16#bd8f9666), (dw:=16#3e0bdb4a), (dw:=16#3e37fa0a), (dw:=16#3c819f08), (dw:=16#be86cd15)];
    weights_1_2: ARRAY[1..11] OF EEL.dwREAL := [(dw:=16#3d090a68), (dw:=16#be93b902), (dw:=16#3d9a33a4), (dw:=16#3df1735f), (dw:=16#3d3ce04f), (dw:=16#3e2390fb), (dw:=16#3e5852d3), (dw:=16#bcf6db45), (dw:=16#3d3e1968), (dw:=16#3cee30ba), (dw:=16#3e58a544)];
    weights_1_3: ARRAY[1..11] OF EEL.dwREAL := [(dw:=16#bd982dec), (dw:=16#bdb5ea5d), (dw:=16#3b3d5078), (dw:=16#bd97f26e), (dw:=16#bc97af7c), (dw:=16#bcfd8fa8), (dw:=16#bc30eb28), (dw:=16#bd4e527d), (dw:=16#3d78a460), (dw:=16#3d92946b), (dw:=16#bc42419d)];
    weights_1_4: ARRAY[1..11] OF EEL.dwREAL := [(dw:=16#bc3058d6), (dw:=16#bd4f4a0b), (dw:=16#bd32229b), (dw:=16#3bd0b607), (dw:=16#bc42c452), (dw:=16#bc248ff6), (dw:=16#bd08220e), (dw:=16#bd8c0b17), (dw:=16#3cc4fb2e), (dw:=16#3d070c02), (dw:=16#3e0c8c2c)];
    weights_1_5: ARRAY[1..11] OF EEL.dwREAL := [(dw:=16#bbc1c3c4), (dw:=16#3dc4e8ec), (dw:=16#3e33c873), (dw:=16#3c01b44c), (dw:=16#3d7b4325), (dw:=16#be3c584f), (dw:=16#be18f3a4), (dw:=16#3ced8499), (dw:=16#b7cb948b), (dw:=16#bd88c20f), (dw:=16#3db67f86)];
    weights_1_6: ARRAY[1..11] OF EEL.dwREAL := [(dw:=16#bc698d01), (dw:=16#be334d8d), (dw:=16#bdfaa5ca), (dw:=16#3e12c0a8), (dw:=16#3dcb655b), (dw:=16#3d380c64), (dw:=16#3da8a417), (dw:=16#3dfebda3), (dw:=16#bdbafad2), (dw:=16#3e1579e3), (dw:=16#3e2dc8b5)];
    weights_1_7: ARRAY[1..11] OF EEL.dwREAL := [(dw:=16#bdfdeec5), (dw:=16#be108b05), (dw:=16#3d15f678), (dw:=16#bd137f0a), (dw:=16#be77bfec), (dw:=16#3e893b55), (dw:=16#bd1d6f99), (dw:=16#be08c5da), (dw:=16#3dab0651), (dw:=16#bd4ebf13), (dw:=16#3e6f7455)];
    weights_1_8: ARRAY[1..11] OF EEL.dwREAL := [(dw:=16#bba5054b), (dw:=16#3e7112e8), (dw:=16#bea58441), (dw:=16#3dff15ec), (dw:=16#3c8c6252), (dw:=16#3c174648), (dw:=16#3dfbd7a8), (dw:=16#3dfe46fe), (dw:=16#3d39041d), (dw:=16#bdf86927), (dw:=16#bd2dfb8c)];
    weights_1_9: ARRAY[1..11] OF EEL.dwREAL := [(dw:=16#bdce4a81), (dw:=16#3d462171), (dw:=16#bca7a58b), (dw:=16#bde4ad50), (dw:=16#3d9d743c), (dw:=16#be84709a), (dw:=16#3ead85f7), (dw:=16#be446757), (dw:=16#3e1eac10), (dw:=16#bded46ca), (dw:=16#be7f7100)];
    weights_1_10: ARRAY[1..11] OF EEL.dwREAL := [(dw:=16#bbf3940c), (dw:=16#3d76e07e), (dw:=16#3dee92da), (dw:=16#bd6ed284), (dw:=16#3cfaa8e4), (dw:=16#3e453349), (dw:=16#3e60fe93), (dw:=16#bdc81f8a), (dw:=16#3e2c150e), (dw:=16#3b2a7094), (dw:=16#3d04d8db)];
    weights_1_11: ARRAY[1..11] OF EEL.dwREAL := [(dw:=16#3c2ea456), (dw:=16#be5cc7d0), (dw:=16#be01495f), (dw:=16#3da2b611), (dw:=16#bba61fbd), (dw:=16#bc174921), (dw:=16#bdccff71), (dw:=16#3d8e76bb), (dw:=16#bdda23f6), (dw:=16#3e4c6709), (dw:=16#3e54267e)];
    weights_1_12: ARRAY[1..11] OF EEL.dwREAL := [(dw:=16#bbba0d6d), (dw:=16#3d57296b), (dw:=16#bca2ef38), (dw:=16#bcbb4220), (dw:=16#be00f866), (dw:=16#3e35ce4a), (dw:=16#3d233935), (dw:=16#be3a5525), (dw:=16#3e34ea8a), (dw:=16#bd3b4101), (dw:=16#3db98205)];
    weights_1_13: ARRAY[1..11] OF EEL.dwREAL := [(dw:=16#be288f7f), (dw:=16#3e107c1f), (dw:=16#bd06a9b6), (dw:=16#3df78a53), (dw:=16#3dd0120a), (dw:=16#bda45f30), (dw:=16#3c84573b), (dw:=16#bd31215f), (dw:=16#bde424ba), (dw:=16#bb6dbc64), (dw:=16#3df5aa1d)];
    weights_1_14: ARRAY[1..11] OF EEL.dwREAL := [(dw:=16#3e6d2770), (dw:=16#be925a3f), (dw:=16#3d877dbb), (dw:=16#3dcbdf20), (dw:=16#bd1cbb6f), (dw:=16#3dcaf419), (dw:=16#3c1fcb15), (dw:=16#3d34238d), (dw:=16#be222370), (dw:=16#3d922d6d), (dw:=16#3e52bed6)];
    weights_1_15: ARRAY[1..11] OF EEL.dwREAL := [(dw:=16#bd2818bf), (dw:=16#3dd36de6), (dw:=16#be4be647), (dw:=16#bbe297ed), (dw:=16#bde7d4d1), (dw:=16#3cdb5d6a), (dw:=16#3a3cc3b3), (dw:=16#3d8c1707), (dw:=16#be33f862), (dw:=16#3e0a5eb0), (dw:=16#3e3970dc)];
    weights_1_16: ARRAY[1..11] OF EEL.dwREAL := [(dw:=16#bd2de4c0), (dw:=16#3e55d314), (dw:=16#3bddefec), (dw:=16#be1c4ccc), (dw:=16#3bcc198d), (dw:=16#bc2e370e), (dw:=16#bd8cc45f), (dw:=16#be2b38c2), (dw:=16#bdc64216), (dw:=16#bde618b6), (dw:=16#bda99096)];
    weights_1_17: ARRAY[1..11] OF EEL.dwREAL := [(dw:=16#3cfa9b4f), (dw:=16#3e59a614), (dw:=16#bd04af9b), (dw:=16#3e4c9a40), (dw:=16#3ccc4af4), (dw:=16#be6c36f3), (dw:=16#bde3f2a0), (dw:=16#be602fb2), (dw:=16#be6bc7b6), (dw:=16#3e57397d), (dw:=16#3e65633e)];
    weights_1_18: ARRAY[1..11] OF EEL.dwREAL := [(dw:=16#3c9f6b35), (dw:=16#be25f168), (dw:=16#bc605788), (dw:=16#3b2ebd8c), (dw:=16#3dde192a), (dw:=16#3a032587), (dw:=16#bce6481f), (dw:=16#3d75019d), (dw:=16#3d99bc08), (dw:=16#3e1ccf1f), (dw:=16#3cc567bf)];
    weights_1_19: ARRAY[1..11] OF EEL.dwREAL := [(dw:=16#3c5ae91f), (dw:=16#bca2fc5d), (dw:=16#3e3d9ba6), (dw:=16#3da88868), (dw:=16#bca3a2c2), (dw:=16#bd24091a), (dw:=16#bc7c97bf), (dw:=16#3d898dcd), (dw:=16#bd806fe6), (dw:=16#3cda1318), (dw:=16#bdb2aabd)];
    weights_1_20: ARRAY[1..11] OF EEL.dwREAL := [(dw:=16#bd978a2e), (dw:=16#bd657deb), (dw:=16#3d8d460d), (dw:=16#bdc6d92c), (dw:=16#bd77cafc), (dw:=16#bdcb811b), (dw:=16#3d60dfba), (dw:=16#3e056cb5), (dw:=16#bd8c9a7d), (dw:=16#3b6db11f), (dw:=16#bdea71fa)];
    weights_1_21: ARRAY[1..11] OF EEL.dwREAL := [(dw:=16#3e505591), (dw:=16#bdc52d7a), (dw:=16#3e961471), (dw:=16#bd5a30fc), (dw:=16#bd226d01), (dw:=16#be46f4f4), (dw:=16#be242bff), (dw:=16#3e18b963), (dw:=16#bdff5f43), (dw:=16#3d295006), (dw:=16#bbabf622)];
    weights_1_22: ARRAY[1..11] OF EEL.dwREAL := [(dw:=16#bde377d4), (dw:=16#3e382e44), (dw:=16#bdeb328b), (dw:=16#3e88c968), (dw:=16#bdf69508), (dw:=16#be1b73ed), (dw:=16#3ca8f494), (dw:=16#bdeba865), (dw:=16#3df15103), (dw:=16#bea752de), (dw:=16#3d136b89)];
    weights_1_23: ARRAY[1..11] OF EEL.dwREAL := [(dw:=16#bdc41321), (dw:=16#bd5827c4), (dw:=16#be06bd3f), (dw:=16#bc3b4ddd), (dw:=16#bd9cea2c), (dw:=16#3db44fbd), (dw:=16#3da1b3c3), (dw:=16#bdfa1b43), (dw:=16#be166080), (dw:=16#3c83bfaf), (dw:=16#3c8d2086)];
    weights_1_24: ARRAY[1..11] OF EEL.dwREAL := [(dw:=16#3e7288cd), (dw:=16#be6a780c), (dw:=16#3e5e8d2a), (dw:=16#be56126a), (dw:=16#bd358bdf), (dw:=16#3e00949b), (dw:=16#be14b50b), (dw:=16#3e1f9836), (dw:=16#3cbaf9c0), (dw:=16#3d68aaea), (dw:=16#bd481dd7)];
    weights_1_25: ARRAY[1..11] OF EEL.dwREAL := [(dw:=16#3d160fe1), (dw:=16#3c3cbac5), (dw:=16#be0bd625), (dw:=16#3d9487e4), (dw:=16#3e564de0), (dw:=16#bd69ccad), (dw:=16#3e3095d1), (dw:=16#3e01b73f), (dw:=16#be3d5c42), (dw:=16#3ec6596c), (dw:=16#bd06c479)];
    weights_2_1: ARRAY[1..25] OF EEL.dwREAL := [(dw:=16#3ebdc266), (dw:=16#3e9b4227), (dw:=16#3e3e85c2), (dw:=16#3dd95fe4), (dw:=16#3e73b422), (dw:=16#be041dc1), (dw:=16#bd7094e6), (dw:=16#bd617f2b), (dw:=16#3e126a81), (dw:=16#3e30ee4f), (dw:=16#3d55259e), (dw:=16#3df4936d), (dw:=16#bd720a0a), (dw:=16#3ea90383), (dw:=16#3e8fea46), (dw:=16#3e36076c), (dw:=16#3c022e69), (dw:=16#bbb5835a), (dw:=16#3cfca8cf), (dw:=16#3d61cfd6), (dw:=16#3e9f339e), (dw:=16#3e931f10), (dw:=16#3e461ee7), (dw:=16#bc7fe5f7), (dw:=16#3ce83186)];
    weights_2_2: ARRAY[1..25] OF EEL.dwREAL := [(dw:=16#3eaebc80), (dw:=16#bda1b632), (dw:=16#3ebe62e2), (dw:=16#3e9030bc), (dw:=16#3e0e7ca0), (dw:=16#3d0421be), (dw:=16#3ec76c81), (dw:=16#3d51c804), (dw:=16#3ea9ea15), (dw:=16#3e0d627a), (dw:=16#3ecebb6f), (dw:=16#3e83c34f), (dw:=16#bbbebf5c), (dw:=16#3ed80cc3), (dw:=16#be5c4c45), (dw:=16#3e93f9cb), (dw:=16#3e8a9752), (dw:=16#3eac1587), (dw:=16#3ea96e96), (dw:=16#3da67ebf), (dw:=16#3e99c2ae), (dw:=16#be4b57da), (dw:=16#bbd169f7), (dw:=16#3eee5a15), (dw:=16#be71a16d)];
    weights_2_3: ARRAY[1..25] OF EEL.dwREAL := [(dw:=16#3d85a2e5), (dw:=16#be92d920), (dw:=16#bd630690), (dw:=16#bc9b6f2f), (dw:=16#be50b663), (dw:=16#3eaa7347), (dw:=16#3df01ea9), (dw:=16#3e90da13), (dw:=16#3e19deb2), (dw:=16#bd082a93), (dw:=16#3e2943aa), (dw:=16#bcc962cf), (dw:=16#3ebd08a9), (dw:=16#be05aea1), (dw:=16#be4b1a64), (dw:=16#3d47c372), (dw:=16#3f009bf3), (dw:=16#3df7b8db), (dw:=16#3d4ad68a), (dw:=16#3e307a6f), (dw:=16#beaa4969), (dw:=16#be951d28), (dw:=16#bdb646c6), (dw:=16#3e690392), (dw:=16#bea88186)];
    weights_2_4: ARRAY[1..25] OF EEL.dwREAL := [(dw:=16#3e0206f6), (dw:=16#3d7511e7), (dw:=16#be047c61), (dw:=16#3b7b7025), (dw:=16#be1cfd90), (dw:=16#3e83c750), (dw:=16#3e5faea1), (dw:=16#3eb9c070), (dw:=16#3e876d47), (dw:=16#3e453994), (dw:=16#3dbc7912), (dw:=16#3e736704), (dw:=16#3e658091), (dw:=16#3dc4c3bd), (dw:=16#3e394ae6), (dw:=16#3e2c5058), (dw:=16#3d1ed50e), (dw:=16#bd885b2c), (dw:=16#bd872c81), (dw:=16#3e02fb85), (dw:=16#3e53b690), (dw:=16#be756c2b), (dw:=16#3ce1396b), (dw:=16#3ee562c4), (dw:=16#be497c46)];
    weights_2_5: ARRAY[1..25] OF EEL.dwREAL := [(dw:=16#bd818b3c), (dw:=16#bd83191c), (dw:=16#bd8256ca), (dw:=16#3dfecde8), (dw:=16#b8246c26), (dw:=16#3c73d69a), (dw:=16#3d516608), (dw:=16#bcb55b0d), (dw:=16#bd1f13dd), (dw:=16#bd463a1d), (dw:=16#ba733500), (dw:=16#3dafe952), (dw:=16#3ddbec33), (dw:=16#bd93812d), (dw:=16#be017b5e), (dw:=16#bcb5d970), (dw:=16#be1c8853), (dw:=16#bd0aa4e6), (dw:=16#bcb46df9), (dw:=16#bc81ea04), (dw:=16#bbd5e2a4), (dw:=16#3b1e9ea1), (dw:=16#3c08b4b0), (dw:=16#bcc92842), (dw:=16#bc456c28)];
    weights_3_1: ARRAY[1..5] OF EEL.dwREAL := [(dw:=16#3c88a3f4), (dw:=16#be3fa499), (dw:=16#3c178f4b), (dw:=16#bd05d5be), (dw:=16#3b71cc1c)];
    weights_3_2: ARRAY[1..5] OF EEL.dwREAL := [(dw:=16#be3e5c2d), (dw:=16#3e7bdac0), (dw:=16#3e81a53d), (dw:=16#3ec66d49), (dw:=16#bc54ee1d)];
    weights_3_3: ARRAY[1..5] OF EEL.dwREAL := [(dw:=16#beb11cc1), (dw:=16#3f024583), (dw:=16#3ea70712), (dw:=16#3ddb8815), (dw:=16#bde5f921)];
    weights_3_4: ARRAY[1..5] OF EEL.dwREAL := [(dw:=16#bdc23653), (dw:=16#3ea7b0b7), (dw:=16#3e35fb4b), (dw:=16#bc3c1832), (dw:=16#bbfdd944)];
    weights_3_5: ARRAY[1..5] OF EEL.dwREAL := [(dw:=16#3e5dd4f6), (dw:=16#3d463a4c), (dw:=16#3d22a2f7), (dw:=16#be81f6b3), (dw:=16#3d548243)];
    weights_3_6: ARRAY[1..5] OF EEL.dwREAL := [(dw:=16#3d75a771), (dw:=16#3dac320e), (dw:=16#be4400bd), (dw:=16#3e13c46e), (dw:=16#3b4dec50)];
    weights_3_7: ARRAY[1..5] OF EEL.dwREAL := [(dw:=16#be0bb40a), (dw:=16#3edc43cc), (dw:=16#3ea958d4), (dw:=16#3eb17e7e), (dw:=16#bc27a9e2)];
    weights_3_8: ARRAY[1..5] OF EEL.dwREAL := [(dw:=16#bee73156), (dw:=16#3da4fb95), (dw:=16#3f264dea), (dw:=16#3ee1b1a1), (dw:=16#bd0225fc)];
    weights_3_9: ARRAY[1..5] OF EEL.dwREAL := [(dw:=16#a996fe99), (dw:=16#bdea618a), (dw:=16#bd35be55), (dw:=16#3e3d650b), (dw:=16#80000023)];
    weights_3_10: ARRAY[1..5] OF EEL.dwREAL := [(dw:=16#ad0d308c), (dw:=16#ba1ce3fc), (dw:=16#a6fb0b24), (dw:=16#a38d5af9), (dw:=16#3d500340)];
    weights_3_11: ARRAY[1..5] OF EEL.dwREAL := [(dw:=16#f6856a1), (dw:=16#b9803b60), (dw:=16#b3601fe0), (dw:=16#b103a2d7), (dw:=16#3d1bc479)];
    weights_3_12: ARRAY[1..5] OF EEL.dwREAL := [(dw:=16#be3faa3f), (dw:=16#3ebe9413), (dw:=16#3ed8d30d), (dw:=16#bc349b48), (dw:=16#bc587680)];
    weights_3_13: ARRAY[1..5] OF EEL.dwREAL := [(dw:=16#ba8495a7), (dw:=16#bc1c1d36), (dw:=16#bb35bda7), (dw:=16#bb941cc9), (dw:=16#3d901a20)];
    weights_3_14: ARRAY[1..5] OF EEL.dwREAL := [(dw:=16#b45ab72d), (dw:=16#bc51549d), (dw:=16#3beb5968), (dw:=16#af63357b), (dw:=16#3dbef7d0)];
    weights_3_15: ARRAY[1..5] OF EEL.dwREAL := [(dw:=16#be783a0e), (dw:=16#3edcf1fd), (dw:=16#3eb2f997), (dw:=16#3e7d5dec), (dw:=16#bcc26646)];
    weights_3_16: ARRAY[1..5] OF EEL.dwREAL := [(dw:=16#2f829a60), (dw:=16#8000045d), (dw:=16#80000000), (dw:=16#80000000), (dw:=16#b3095bfd)];
    weights_3_17: ARRAY[1..5] OF EEL.dwREAL := [(dw:=16#bd8f552a), (dw:=16#3e892b72), (dw:=16#3de40b70), (dw:=16#3dfdfd5d), (dw:=16#bbd063ca)];
    weights_3_18: ARRAY[1..5] OF EEL.dwREAL := [(dw:=16#3123ae87), (dw:=16#11ba2a13), (dw:=16#b409119a), (dw:=16#a60e49f3), (dw:=16#b15266b0)];
    weights_3_19: ARRAY[1..5] OF EEL.dwREAL := [(dw:=16#bea11a26), (dw:=16#3e327abe), (dw:=16#3ec95ed6), (dw:=16#3e9d5faa), (dw:=16#bccbdca5)];
    weights_3_20: ARRAY[1..5] OF EEL.dwREAL := [(dw:=16#a9bfab3c), (dw:=16#8000006a), (dw:=16#80000c70), (dw:=16#98c67e2a), (dw:=16#0)];
    weights_out_1: ARRAY[1..20] OF EEL.dwREAL :=[(dw:=16#bdb04ee6), (dw:=16#3e80c905), (dw:=16#3ee771ca), (dw:=16#3e1303a1), (dw:=16#be8fe765), (dw:=16#bdfa3a61), (dw:=16#3e4bd6c9), (dw:=16#3f05c546), (dw:=16#3d64e793), (dw:=16#bb6c236f), (dw:=16#bba9bcb2), (dw:=16#3e7876f0), (dw:=16#3d1c4119), (dw:=16#bd205805), (dw:=16#3ec1db69), (dw:=16#80c124c8), (dw:=16#3de152f9), (dw:=16#32541b0a), (dw:=16#3ebb7767), (dw:=16#b5c02e34)];
END_VAR

(* get inputs *)
input[1] := in_1;
input[2] := in_2;
input[3] := in_3;
input[4] := in_4;
input[5] := in_5;
input[6] := in_6;
input[7] := in_7;
input[8] := in_8;
input[9] := in_9;
input[10] := in_10;
input[11] := in_11;

(* MLP inference *)
EEL.CallANN(ANN:=MLP);

(* set outputs *)
out_1 := out_neurons[1].output;

END_FUNCTION_BLOCK
